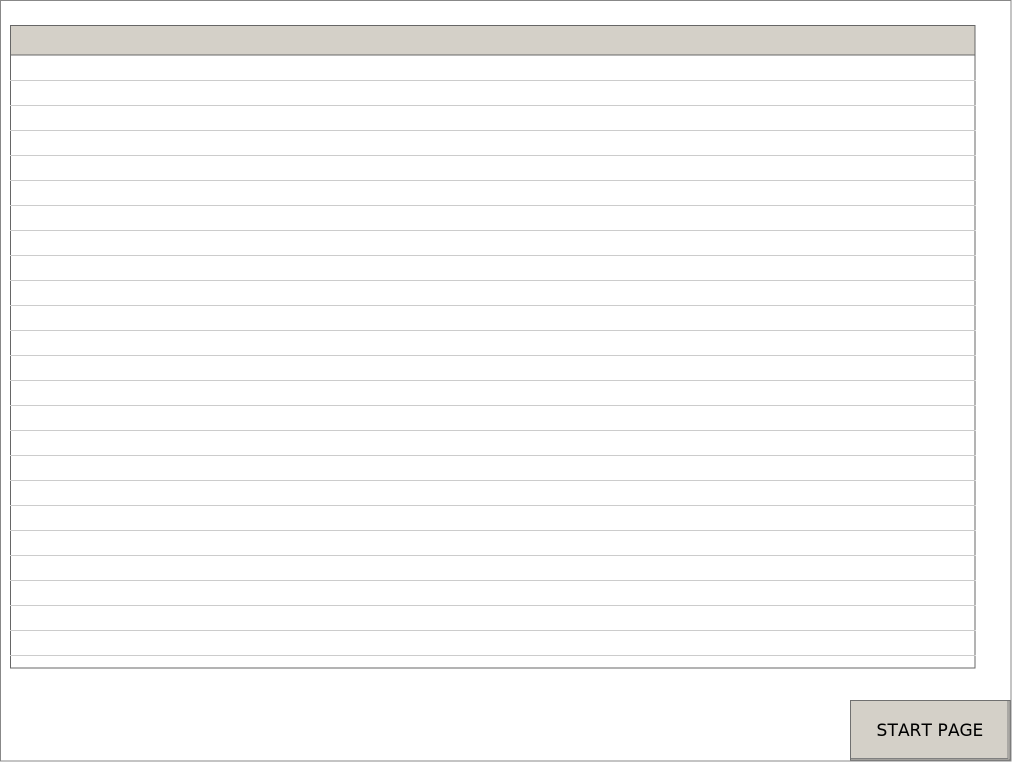
VISUALIZATION HmiEtherCatDiagnostic  // 1012x762
    Button (850,700 160x60), "START PAGE"
        OnMouseClick: change screen: HmiStartPage
    Table (10,25 965x643), data array: fbDiagnosticEtherCAT.stEcTerminalDiagInfo
        p3854506369: fbDiagnosticEtherCAT.stEcTerminalDiagInfo[INDEX].nAddr
        p1892666644: fbDiagnosticEtherCAT.stEcTerminalDiagInfo[INDEX].sType
        p338671338: fbDiagnosticEtherCAT.stEcTerminalDiagInfo[INDEX].sName
        p2170511999: fbDiagnosticEtherCAT.stEcTerminalDiagInfo[INDEX].sTerminalStatus
END_VISUALIZATION

(* stored: Version 1.1.0.1
   Visu HmiEtherCatDiagnostic: Id {0e1114d6-0961-4aea-9d50-3a109c395bb1} *)
